TYPE LogEvent :
STRUCT
	timestamp : Tc2_Utilities.TimeStruct;
	level : LogLevel;
	logger : T_MaxString;
	message : T_MaxString;
END_STRUCT
END_TYPE

(* stored: Version 1.1.0.1
   DUT LogEvent: Id {d23894b2-6075-4807-9e06-8026e94bffa3} *)
